// TIA Portal V20 export
DATA_BLOCK "DB_Marrige"   // DB10
{ S7_Optimized_Access := 'TRUE' }
// stored: AutoNumber false, MemoryReserve 100
   VAR
      Functional_Tests_Panels : Array[0..31] of "Functional_Test";
      Got_Married { S7_SetPoint := 'True'} : Bool;
      Serial_Number : String[17];
   END_VAR
BEGIN
   Functional_Tests_Panels[0].Panel_Number := 0;
   Functional_Tests_Panels[1].Panel_Number := 1;
   Functional_Tests_Panels[2].Panel_Number := 2;
   Functional_Tests_Panels[3].Panel_Number := 3;
   Functional_Tests_Panels[4].Panel_Number := 4;
   Functional_Tests_Panels[5].Panel_Number := 5;
   Functional_Tests_Panels[6].Panel_Number := 6;
   Functional_Tests_Panels[7].Panel_Number := 7;
   Functional_Tests_Panels[8].Panel_Number := 8;
   Functional_Tests_Panels[9].Panel_Number := 9;
   Functional_Tests_Panels[10].Panel_Number := 10;
   Functional_Tests_Panels[11].Panel_Number := 11;
   Functional_Tests_Panels[12].Panel_Number := 12;
   Functional_Tests_Panels[13].Panel_Number := 13;
   Functional_Tests_Panels[14].Panel_Number := 14;
   Functional_Tests_Panels[15].Panel_Number := 15;
   Functional_Tests_Panels[16].Panel_Number := 16;
   Functional_Tests_Panels[17].Panel_Number := 17;
   Functional_Tests_Panels[18].Panel_Number := 18;
   Functional_Tests_Panels[19].Panel_Number := 19;
   Functional_Tests_Panels[20].Panel_Number := 20;
   Functional_Tests_Panels[21].Panel_Number := 21;
   Functional_Tests_Panels[22].Panel_Number := 22;
   Functional_Tests_Panels[23].Panel_Number := 23;
   Functional_Tests_Panels[24].Panel_Number := 24;
   Functional_Tests_Panels[25].Panel_Number := 25;
   Functional_Tests_Panels[26].Panel_Number := 26;
   Functional_Tests_Panels[27].Panel_Number := 27;
   Functional_Tests_Panels[28].Panel_Number := 28;
   Functional_Tests_Panels[29].Panel_Number := 29;
   Functional_Tests_Panels[30].Panel_Number := 30;
   Functional_Tests_Panels[31].Panel_Number := 31;
END_DATA_BLOCK
